PROGRAM analogSignals_ex01
VAR
	Frawsensor		: REAL;
	fScaledvalue	: real;
	
	LIN_TRAFO 		: FB_Scale;
END_VAR

LIN_TRAFO(
	fIN:= frawsensor, 
	fIN_min:= 4, 
	fIN_max:= 20, 
	fOUT_min:= 0, 
	fOUT_max:= 100, 
	fOUT=> fScaledvalue);

END_PROGRAM

(* stored: Version 1.1.0.1
   POU analogSignals_ex01: Id {f4996adb-45ed-48e9-9127-d8c4365a7cab}, SpecialFunc None *)
